// TwinCAT 3 PLC project project_
// ProgramVersion: 3.1.4023.0
// libraries:
//   Tc2_Standard, * (Beckhoff Automation GmbH)
//   Tc2_System, * (Beckhoff Automation GmbH)
//   Tc3_Module, * (Beckhoff Automation GmbH)
// project tree:
//   / PlcTask.TcTTO
//   POUs/ MAIN.TcPOU
// real-time tasks:
//   TASK PlcTask: cycle T#10ms, priority 20, ADS port 350

CONFIGURATION project_
    RESOURCE PLC ON TwinCAT3
        TASK PlcTask(INTERVAL := T#10ms, PRIORITY := 20);
        PROGRAM MAIN WITH PlcTask : MAIN;
    END_RESOURCE
END_CONFIGURATION

// ---- POUs/MAIN.TcPOU
PROGRAM MAIN
VAR
	MyBoolean : BOOL;
	
	bRunMath : BOOL;
	
	iValue1 : DINT := 20;
	iValue2 : DINT;
	
	i : INT;
	j : INT;
	c : DINT;
	
	sMyString : STRING;
	sMyNumString : STRING[255];
	
	i_Num_from_arr : DINT;
	i_len_arr_B : INT;
	arr_A : ARRAY [0..10] OF DINT;
	arr_B : ARRAY [0..4] OF DINT :=[20, 40, 60 ,80, 100];
	
	// timers
	fb_My_timer : TON;
	// tiggers
	fb_my_trigger : R_TRIG; // Counter 
	
	// Timer
	fb_MI1_Timer_Increase_Speed: TON;
	
	// Speed setup
	f_MI1_Initial_Speed: REAL := 20;
	f_MI1_Constant_Speed: REAL := 60;
	f_MI1_Max_Speed : REAL := 120;
END_VAR

VAR_OUTPUT
	// Speed Output
	f_MI1_Speed: REAL;
END_VAR


f_MI1_Speed:= f_MI1_Initial_Speed;

IF MyBoolean THEN
	REPEAT
		fb_MI1_Timer_Increase_Speed(
			IN:=MyBoolean,
			PT:= T#20S);
		IF fb_MI1_Timer_Increase_Speed.Q THEN
			f_MI1_Speed := f_MI1_Speed + f_MI1_Initial_Speed;
		END_IF
		
	UNTIL 
		f_MI1_Speed > 120 
	END_REPEAT
	
END_IF

END_PROGRAM
